KUKA KRL program: MatlabControl.src, MatLabControl.dat

--- MatlabControl.src ---
&ACCESS RVP
&REL 4
DEF MatlabControl()
    DECL INT I

    WAIT FOR $MOVE_ENABLE

    ; Safe init - resets defaults
    BAS(#INITMOV,0)

    ; Set safe initial velocities + accelerations (100%)
    FOR I = 1 TO 6
        $VEL_AXIS[I] = 100
        $ACC_AXIS[I] = 100
    ENDFOR

    ; Safe init for the magnetic command path
    magnetic_cmd = FALSE
    vacuum_cmd = FALSE
    $OUT[25] = FALSE
    $OUT[24] = FALSE

    PTP XHOME

    ; Main loop
    LOOP
        ; Mirror the MATLAB magnetic BOOL command to the physical output.
        ; This keeps KUKAVARPROXY writes on a simple global variable.
        $OUT[25] = magnetic_cmd
        $OUT[24] = vacuum_cmd

        IF $MOVE_ENABLE AND move_trigger THEN
            ; fast move (100%)
            FOR I = 1 TO 6
                $VEL_AXIS[I] = 100
                $ACC_AXIS[I] = 100
            ENDFOR

            ; Tiny settle time for motion planner
            WAIT SEC 0.02

            PTP target_pos
            move_trigger = FALSE
        ENDIF

        WAIT SEC 0.01
    ENDLOOP
END

--- MatLabControl.dat ---
&ACCESS RVP
&REL 4
DEFDAT  MATLABCONTROL PUBLIC

DECL GLOBAL POS target_pos={X 509.876,Y 339.917,Z 552.366,A 0.0,B 90.0000,C 0.0}
DECL GLOBAL BOOL move_trigger=TRUE
DECL GLOBAL BOOL magnetic_cmd=FALSE
DECL GLOBAL BOOL vacuum_cmd=FALSE

ENDDAT
